FUNCTION_BLOCK OF_E_TOF (* standard timer function block (off-delay timing) *)
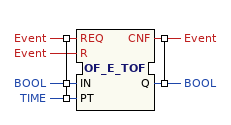
  EVENT_INPUT
    REQ WITH IN, PT; (* Normal Execution Request *)
    R; (* Reset *)
  END_EVENT
  EVENT_OUTPUT
    CNF WITH Q; (* Execution Confirmation *)
  END_EVENT
  VAR_INPUT
    IN : BOOL; (* Input *)
    PT : TIME; (* Process time *)
  END_VAR
  VAR_OUTPUT
    Q : BOOL; (* Output *)
  END_VAR
END_FUNCTION_BLOCK
